# EPICS autosave request: support/ip-2-10/ipApp/Db/LakeShore340.req
# FILE... LakeShore340.req
$(P)LS340:$(Q):Gain_set.VAL
$(P)LS340:$(Q):Rset_set.VAL
$(P)LS340:$(Q):Rate_set.VAL
$(P)LS340:$(Q):RampR_set.VAL
$(P)LS340:$(Q):Ramp_on.VAL
$(P)LS340:$(Q):wr_SP.VAL
$(P)LS340:$(Q):Units_sel.VAL
$(P)LS340:$(Q):Input_sel.VAL
$(P)LS340:$(Q):HeatRg.VAL
$(P)LS340:$(Q):read.SCAN
$(P)LS340:$(Q):rd_rdat_scalc.SCAN
